Staubli VAL3: cycle.pjx

--- cycle.pjx ---
Parameters version=s7.8.3 stackSize=5000 millimeterUnit=true
Program file=_tcycle.pgx
Program file=_tPLC.pgx
Program file=_WatchDog.pgx
Program file=checkIoBus.pgx
Program file=isStopped.pgx
Program file=PowerOn.pgx
Program file=save.pgx
Program file=start.pgx
Program file=stop.pgx
Program file=wizard.pgx
Data file=cycle.dtx
Library alias=data path=Disk://SaveData/SaveData.pjx
Library alias=io path=Disk://io/io.pjx
Library alias=use path=Disk://public_temp/userPage/USERPAGE.pjx

--- cycle.dtx ---
mdesc mNomSpeed
bool bIspower
public bool bIsEstop
num nWorkingStatus
num nWorkingMode
bool bConnected
public bool bCycle
public bool bPause
public bool bIsHome
public bool bRobotErr
public bool bIsRemote
public bool bConnected_Plc
string sIoBusStatus
num nJishu
num x_nResult
public bool bIsReady
string sMenu
num nPage

--- _tcycle.pgx ---
public program _tcycle()
begin
  while true

  endWhile
end

--- _tPLC.pgx ---
public program _tPLC()
  local bool l_bContinue
  local bool l_bStopStatus
begin
  while true

    io:dOutIsReady=(bIsHome and bIsRemote and !bIsEstop and !bRobotErr and !bCycle)
    if io:dOutIsReady==true
      bIsReady=true
    endIf

    //远程自动上电
    if io:dInStart==true
      if taskStatus("cycle")==-1 and bIsReady==true
        bCycle=true
        call PowerOn(l_bContinue)
        if l_bContinue==true
          taskCreate "cycle",100,_tcycle()
          wait(taskStatus("cycle")==1)
        else
          bCycle=false
        endIf
      endIf
      endIf

    if bCycle==true
      call isStopped(l_bStopStatus)
    endIf

  endWhile
end

--- _WatchDog.pgx ---
public program _WatchDog()
  local bool l_bConnected
begin
  while true

    bIspower=isPowered()
    bIsEstop=(esStatus()==2)
//    if abs(herej()-data:jJhome)<{2,2,2,2,2,2}
//      data:bHome=true
//    else
//      data:bHome=false
//    endIf

    //检查通信状况
    nWorkingMode=workingMode(nWorkingStatus)
    call checkIoBus(l_bConnected)
    bConnected_Plc=l_bConnected
    delay(0)
  endWhile
end

--- checkIoBus.pgx ---
public program checkIoBus(bool& x_bBool)
  local num l_nStatus
  local num i
begin
  x_bBool=true
  //check bus status
  l_nStatus=ioBusStatus(sIoBusStatus)
  nJishu=size(sIoBusStatus)
  for i=0 to size(sIoBusStatus)-1
    //是否找到了相应的APLICOM端口
    if left(sIoBusStatus[i],1)!="0"
      x_bBool=false
      return
    endIf
  endFor
end

--- isStopped.pgx ---
public program isStopped(bool& x_bBool)
begin
  //
  if workingMode()!=4
    logMsg("机器人有报警,循环停止")
    return
  endIf

  if io:dInStop==true
    logMsg("机器人程序停止")
    return
  endIf


end

--- PowerOn.pgx ---
public program PowerOn(bool& x_bBool)
begin
  //
  x_bBool=false
  if workingMode()==4
    if isPowered()==false and esStatus()!=2
      autoConnectMove(true)
      enablePower()
      delay(1)
      x_bBool=true
    endIf
  endIf

end

--- save.pgx ---
public program save(num x_nRetrun)
begin
  x_nRetrun=data:libSave()
end

--- wizard.pgx ---
public program wizard()
  local num l_nSelect
  local bool l_bSelect
begin
  l_nSelect=0
  cls()
  while l_nSelect<3
    switch l_nSelect
      case 0
        call use:typeMenu(8,">>")
        call use:typeMenu(7,"<<")
        gotoxy(1,1)
        put("1")
        do
          nPage=getKey()
          if(nPage==278)
            l_nSelect=l_nSelect+1
            l_bSelect=true
          elseIf(nPage==277)
            l_nSelect=5
            return
          endIf
        until l_bSelect==true
      break
      case 1
        call use:typeMenu(8,">>")
        call use:typeMenu(7,"<<")
        gotoxy(1,1)
        put("2")
        do
          nPage=getKey()
          if(nPage==278)
            l_nSelect=l_nSelect+1
            l_bSelect=true
          elseIf(nPage==277)
            l_nSelect=l_nSelect-1
            l_bSelect=true
          endIf
        until l_bSelect==true
      break
      case 2
        call use:typeMenu(8,">>")
        call use:typeMenu(7,"<<")
        gotoxy(1,1)
        put("3")
        do
          nPage=getKey()
          if(nPage==278)
            l_nSelect=l_nSelect+1
            l_bSelect=true
          elseIf(nPage==277)
            l_nSelect=l_nSelect-1
            l_bSelect=true
          endIf
        until l_bSelect==true
      break
      case 3
      break
      case 4
      break
    endSwitch
  endWhile
end
